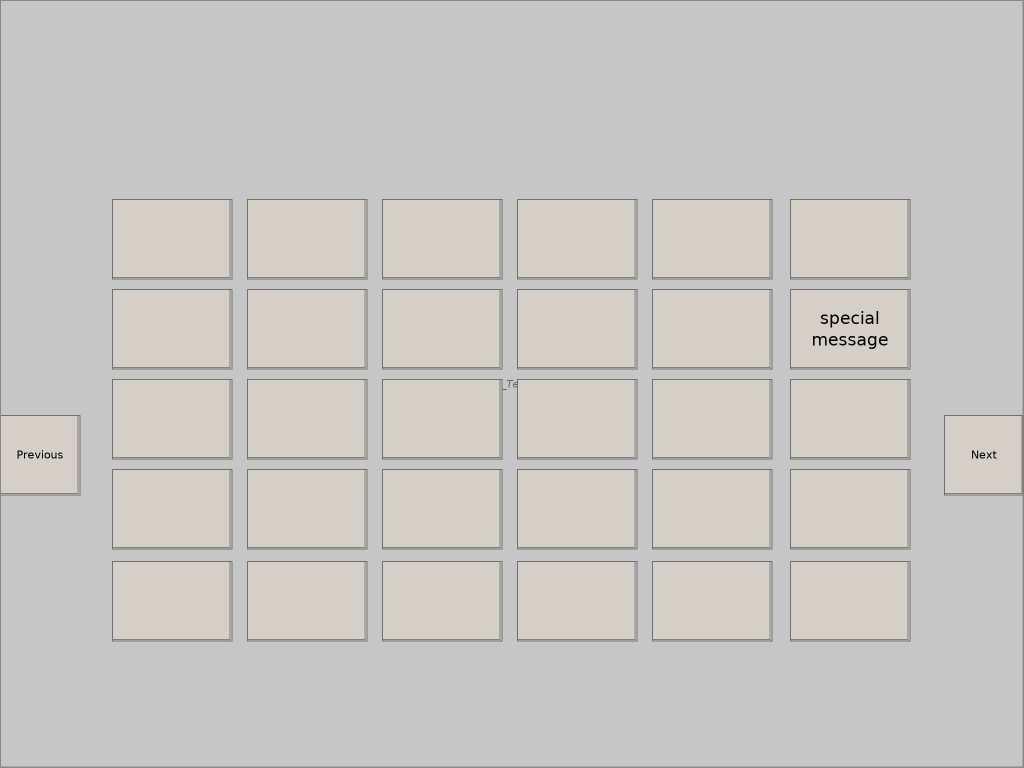
VISUALIZATION SS_10_MenuScreen_3  // 1024x768
    Frame (0,0 1024x768)
        shows SS_91_Template(header := HMIData.hmiHeader)
    Button (112,199 120x80), text list: ''
    Button (247,199 120x80), text list: ''
    Button (382,199 120x80), text list: ''
    Button (517,199 120x80), text list: ''
    Button (652,199 120x80), text list: ''
    Button (790,199 120x80), text list: ''
    Button (112,289 120x80), text list: ''
    Button (247,289 120x80), text list: ''
    Button (382,289 120x80), text list: ''
    Button (517,289 120x80), text list: ''
    Button (652,289 120x80), text list: ''
    Button (790,289 120x80), "special message", text list: ''
        OnMouseClick: change screen: SS_12_AlarmsTest
    Button (112,379 120x80), text list: ''
    Button (247,379 120x80), text list: ''
    Button (382,379 120x80), text list: ''
    Button (517,379 120x80), text list: ''
    Button (652,379 120x80), text list: ''
    Button (790,379 120x80), text list: ''
    Button (112,469 120x80), text list: ''
    Button (247,469 120x80), text list: ''
    Button (382,469 120x80), text list: ''
    Button (517,469 120x80), text list: ''
    Button (652,469 120x80), text list: ''
    Button (790,469 120x80), text list: ''
    Button (112,561 120x80), text list: ''
    Button (247,561 120x80), text list: ''
    Button (382,561 120x80), text list: ''
    Button (517,561 120x80), text list: ''
    Button (652,561 120x80), text list: ''
    Button (790,561 120x80), text list: ''
    Group (0,415 1024x80)
        Button (0,0 80x80), "Previous"
            OnMouseClick: change screen: SS_10_MenuScreen_2
        Button (944,0 80x80), "Next"
            OnMouseClick: change screen: SS_10_MenuScreen
END_VISUALIZATION

(* stored: Version 1.1.0.1, ProductVersion 3.1.4024.12
   Visu SS_10_MenuScreen_3: Id {73b9ea03-2c91-46d6-a0f2-36ef36d02056} *)
